// TIA Portal project "PLC_IHM" (V17)

(* hardware
DEVICE "HMI_1"  KTP400 Comfort
   slot 0: "HMI_1"  KTP400 Comfort  6AV2 124-2DC01-0AX0  16.0.0.0
   slot 1: "HMI_RT_1"  KTP400 Comfort  6AV2 124-2DC01-0AX0  16.0.0.0
   slot 5: "HMI_1.IE_CP_1"  PROFINET Interface  16.0.0.0
      slot 1: "PROFINET Interface_1"  PROFINET Interface
         slot 1: "Port_1"  Port
   slot 7: "HMI_1.MPI/DP_CP_1"  MPI/DP Interface  16.0.0.0
DEVICE "S7-1200 station_1"  S7-1200 Station
   slot 0: "Rack_0"  S7-1200 Rack  Rack  V1.0
   slot 1: "PLC_1"  CPU 1211C DC/DC/Rly  6ES7 211-1HE40-0XB0  V4.5
*)

// ===== PLC "PLC_1"  CPU 1211C DC/DC/Rly =====

VAR_GLOBAL   // PLC tag table "Default tag table"
   "Tag_1" AT %I0.0 : Bool;
   "Tag_3" AT %I0.1 : Bool;
   "Tag_5" AT %I0.2 : Bool;
   "Tag_8" AT %I0.3 : Bool;
   "Tag_9" AT %I0.4 : Bool;
   "CPLUS" AT %Q0.0 : Bool;
   "CMOINS" AT %Q0.1 : Bool;
   "MPLUS" AT %Q0.2 : Bool;
   "MMOINS" AT %Q0.3 : Bool;
   "IHM_TEST_Q0" AT %M0.0 : Bool;
   "IHM_TEST_Q1" AT %M0.1 : Bool;
   "IHM_TEST_Q2" AT %M0.2 : Bool;
   "IHM_TEST_Q3" AT %M0.3 : Bool;
   "X0" AT %M1.0 : Bool;
   "X2" AT %M1.1 : Bool;
   "X3" AT %M1.2 : Bool;
   "X4" AT %M1.3 : Bool;
   "X5" AT %M1.4 : Bool;
   "X6" AT %M1.5 : Bool;
   "X7" AT %M1.6 : Bool;
   "DCY" AT %M2.0 : Bool;
   "C1" AT %M2.1 : Bool;
   "C2" AT %M2.2 : Bool;
   "C3" AT %M2.3 : Bool;
   "DECHARGE" AT %M2.4 : Bool;
   "HAUT" AT %M2.5 : Bool;
   "BAS" AT %M2.6 : Bool;
   "X1" AT %M2.7 : Bool;
   "FIN_TEMPO" AT %M3.0 : Bool;
   "MOVE_X_PIECE" AT %MW20 : Int;
   "MOVE_Y_PIECE" AT %MW4 : Int;
   "SendInitParam" AT %M3.1 : Bool;
   "SendInitMemo" AT %M3.2 : Bool;
   "MOVE_X_CHARIOT" AT %MW6 : Int;
   "MOVE_Y_CHARIOT" AT %MW8 : Int;
   "MOVE_X_CORDON" AT %MW10 : Int;
   "MOVE_Y_CORDON" AT %MW12 : Int;
   "tempoTime" AT %MD30 : Time;
   "CompteurPiece" AT %MW24 : Int;
   "MemoI0" AT %M30.0 : Bool;
   "MemoI1" AT %M30.1 : Bool;
   "MemoI2" AT %M30.2 : Bool;
   "MemoI3" AT %M30.3 : Bool;
   "Tempo_Int_To_Time" AT %MD34 : Time;
   "Tempo_Int" AT %MW26 : Int;
   "Tempo_Time_To_Int" AT %MW28 : Int;
END_VAR

// folder: System blocks/Program resources

DATA_BLOCK "TEMPO"   // DB1
{ S7_Optimized_Access := 'TRUE' }
AUTHOR : Simatic
FAMILY : IEC
NAME : IEC_TMR
VERSION : 1.0
// stored: InstanceOfName IEC_TIMER
"IEC_TIMER"
BEGIN
END_DATA_BLOCK

// folder: (top level)

FUNCTION "TestInputOutput" : Void   // FC1, LAD
{ S7_Optimized_Access := 'TRUE' }
VERSION : 0.1
BEGIN

REGION Network 1: I0 alumme Q0
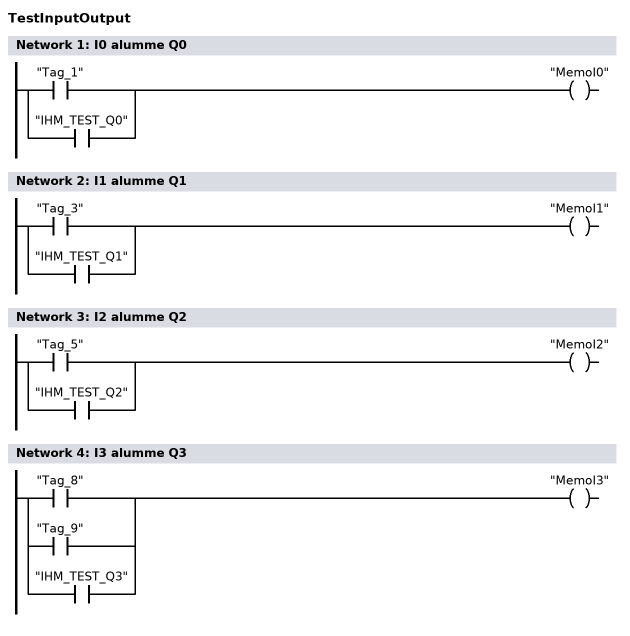
   RUNG wire#powerrail
      Contact( "Tag_1" )
      wire#w1
      Coil( "MemoI0" )
   END_RUNG
   RUNG wire#powerrail
      Contact( "IHM_TEST_Q0" )
   END_RUNG wire#w1
   // the same network as SCL:
   "MemoI0" := "Tag_1" OR "IHM_TEST_Q0";
END_REGION

REGION Network 2: I1 alumme Q1
   RUNG wire#powerrail
      Contact( "Tag_3" )
      wire#w1
      Coil( "MemoI1" )
   END_RUNG
   RUNG wire#powerrail
      Contact( "IHM_TEST_Q1" )
   END_RUNG wire#w1
   // the same network as SCL:
   "MemoI1" := "Tag_3" OR "IHM_TEST_Q1";
END_REGION

REGION Network 3: I2 alumme Q2
   RUNG wire#powerrail
      Contact( "Tag_5" )
      wire#w1
      Coil( "MemoI2" )
   END_RUNG
   RUNG wire#powerrail
      Contact( "IHM_TEST_Q2" )
   END_RUNG wire#w1
   // the same network as SCL:
   "MemoI2" := "Tag_5" OR "IHM_TEST_Q2";
END_REGION

REGION Network 4: I3 alumme Q3
   RUNG wire#powerrail
      Contact( "Tag_8" )
      wire#w1
      Coil( "MemoI3" )
   END_RUNG
   RUNG wire#powerrail
      Contact( "Tag_9" )
   END_RUNG wire#w1
   RUNG wire#powerrail
      Contact( "IHM_TEST_Q3" )
   END_RUNG wire#w1
   // the same network as SCL:
   "MemoI3" := "Tag_8" OR "Tag_9" OR "IHM_TEST_Q3";
END_REGION
END_FUNCTION

FUNCTION "BAIN_DEGRESSAGE" : Void   // FC2, LAD
{ S7_Optimized_Access := 'TRUE' }
VERSION : 0.1
BEGIN

REGION Network 1: X0
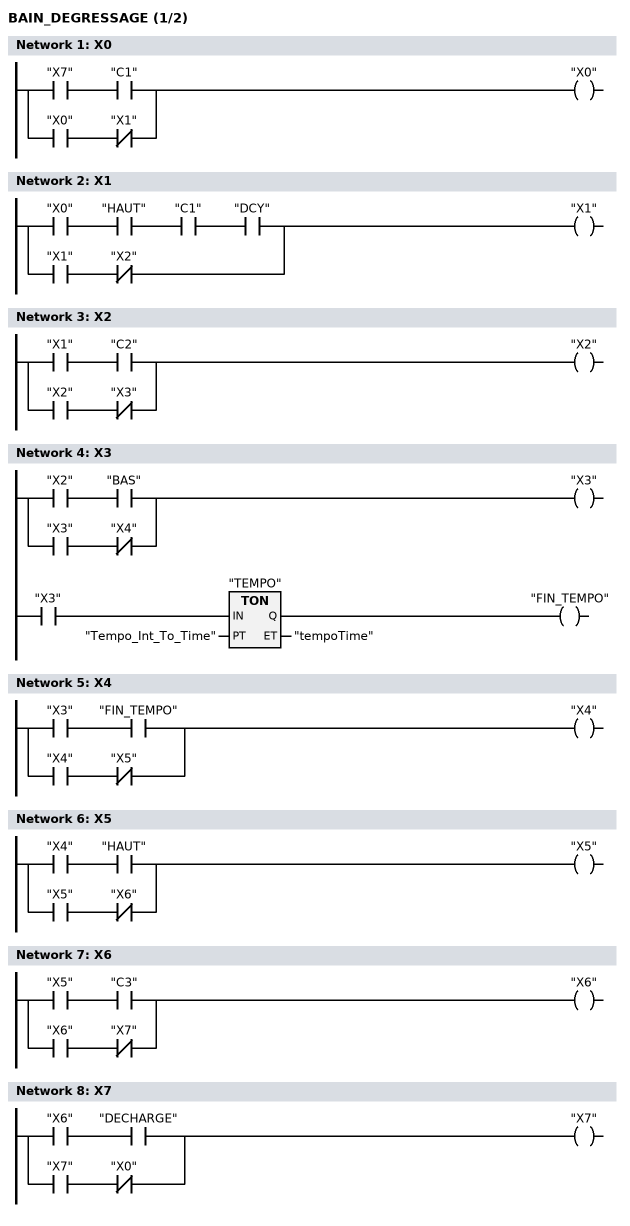
   RUNG wire#powerrail
      Contact( "X7" )
      Contact( "C1" )
      wire#w1
      Coil( "X0" )
   END_RUNG
   RUNG wire#powerrail
      Contact( "X0" )
      I_Contact( "X1" )
   END_RUNG wire#w1
   // the same network as SCL:
   "X0" := ("X7" AND "C1") OR ("X0" AND NOT "X1");
END_REGION

REGION Network 2: X1
   RUNG wire#powerrail
      Contact( "X0" )
      Contact( "HAUT" )
      Contact( "C1" )
      Contact( "DCY" )
      wire#w1
      Coil( "X1" )
   END_RUNG
   RUNG wire#powerrail
      Contact( "X1" )
      I_Contact( "X2" )
   END_RUNG wire#w1
   // the same network as SCL:
   "X1" := ("X0" AND "HAUT" AND "C1" AND "DCY") OR ("X1" AND NOT "X2");
END_REGION

REGION Network 3: X2
   RUNG wire#powerrail
      Contact( "X1" )
      Contact( "C2" )
      wire#w1
      Coil( "X2" )
   END_RUNG
   RUNG wire#powerrail
      Contact( "X2" )
      I_Contact( "X3" )
   END_RUNG wire#w1
   // the same network as SCL:
   "X2" := ("X1" AND "C2") OR ("X2" AND NOT "X3");
END_REGION

REGION Network 4: X3
   "X3" := ("X2" AND "BAS") OR ("X3" AND NOT "X4");
   "TEMPO".TON(IN := "X3", PT := "Tempo_Int_To_Time", ET => "tempoTime");
   "FIN_TEMPO" := "TEMPO".Q;
END_REGION

REGION Network 5: X4
   RUNG wire#powerrail
      Contact( "X3" )
      Contact( "FIN_TEMPO" )
      wire#w1
      Coil( "X4" )
   END_RUNG
   RUNG wire#powerrail
      Contact( "X4" )
      I_Contact( "X5" )
   END_RUNG wire#w1
   // the same network as SCL:
   "X4" := ("X3" AND "FIN_TEMPO") OR ("X4" AND NOT "X5");
END_REGION

REGION Network 6: X5
   RUNG wire#powerrail
      Contact( "X4" )
      Contact( "HAUT" )
      wire#w1
      Coil( "X5" )
   END_RUNG
   RUNG wire#powerrail
      Contact( "X5" )
      I_Contact( "X6" )
   END_RUNG wire#w1
   // the same network as SCL:
   "X5" := ("X4" AND "HAUT") OR ("X5" AND NOT "X6");
END_REGION

REGION Network 7: X6
   RUNG wire#powerrail
      Contact( "X5" )
      Contact( "C3" )
      wire#w1
      Coil( "X6" )
   END_RUNG
   RUNG wire#powerrail
      Contact( "X6" )
      I_Contact( "X7" )
   END_RUNG wire#w1
   // the same network as SCL:
   "X6" := ("X5" AND "C3") OR ("X6" AND NOT "X7");
END_REGION

REGION Network 8: X7
   RUNG wire#powerrail
      Contact( "X6" )
      Contact( "DECHARGE" )
      wire#w1
      Coil( "X7" )
   END_RUNG
   RUNG wire#powerrail
      Contact( "X7" )
      I_Contact( "X0" )
   END_RUNG wire#w1
   // the same network as SCL:
   "X7" := ("X6" AND "DECHARGE") OR ("X7" AND NOT "X0");
END_REGION

REGION Network 9: SORTIE CPLUS
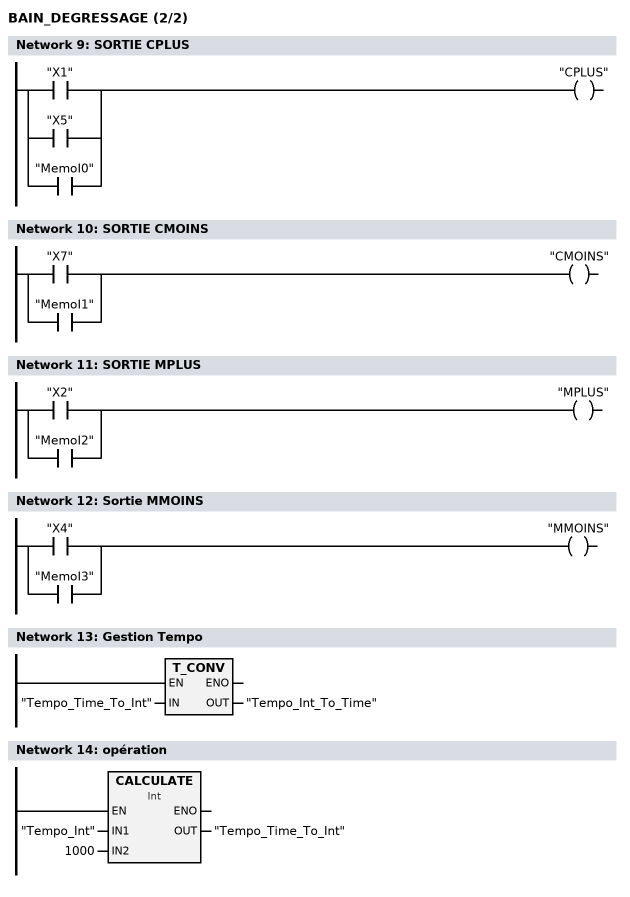
   RUNG wire#powerrail
      Contact( "X1" )
      wire#w1
      Coil( "CPLUS" )
   END_RUNG
   RUNG wire#powerrail
      Contact( "X5" )
   END_RUNG wire#w1
   RUNG wire#powerrail
      Contact( "MemoI0" )
   END_RUNG wire#w1
   // the same network as SCL:
   "CPLUS" := "X1" OR "X5" OR "MemoI0";
END_REGION

REGION Network 10: SORTIE CMOINS
   RUNG wire#powerrail
      Contact( "X7" )
      wire#w1
      Coil( "CMOINS" )
   END_RUNG
   RUNG wire#powerrail
      Contact( "MemoI1" )
   END_RUNG wire#w1
   // the same network as SCL:
   "CMOINS" := "X7" OR "MemoI1";
END_REGION

REGION Network 11: SORTIE MPLUS
   RUNG wire#powerrail
      Contact( "X2" )
      wire#w1
      Coil( "MPLUS" )
   END_RUNG
   RUNG wire#powerrail
      Contact( "MemoI2" )
   END_RUNG wire#w1
   // the same network as SCL:
   "MPLUS" := "X2" OR "MemoI2";
END_REGION

REGION Network 12: Sortie MMOINS
   RUNG wire#powerrail
      Contact( "X4" )
      wire#w1
      Coil( "MMOINS" )
   END_RUNG
   RUNG wire#powerrail
      Contact( "MemoI3" )
   END_RUNG wire#w1
   // the same network as SCL:
   "MMOINS" := "X4" OR "MemoI3";
END_REGION

REGION Network 13: Gestion Tempo
   "Tempo_Int_To_Time" := T_CONV(IN := "Tempo_Time_To_Int");
END_REGION

REGION Network 14: opération
   RUNG wire#powerrail
      { S7_Templates := "SrcType := Int"; S7_Expression := "IN1 * IN2" } Calculate(in1 := "Tempo_Int", in2 := 1000, out => "Tempo_Time_To_Int")
   END_RUNG
   // the same network as SCL:
   "Tempo_Time_To_Int" := "Tempo_Int" * 1000;
END_REGION
END_FUNCTION

FUNCTION "Maintenance" : Void   // FC3, LAD
{ S7_Optimized_Access := 'TRUE' }
VERSION : 0.1
BEGIN

REGION Network 1
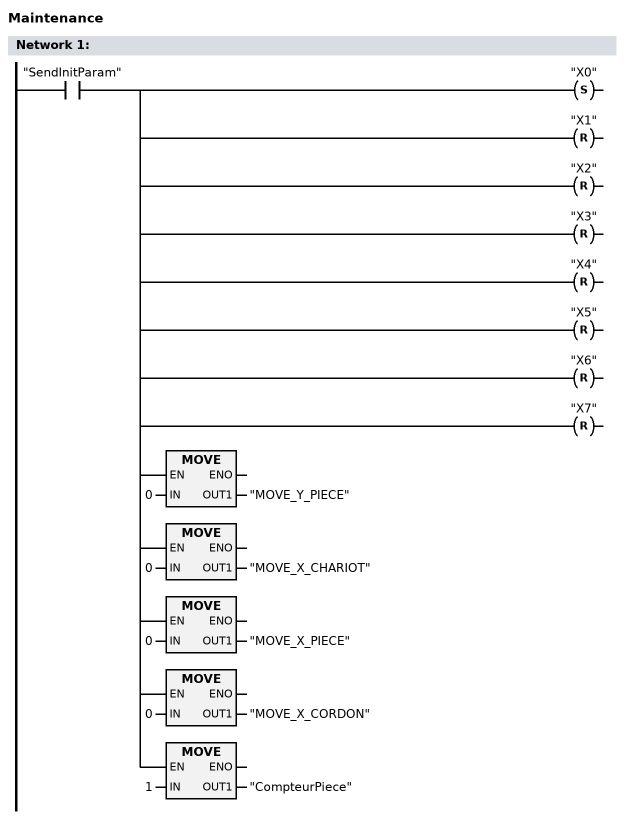
   RUNG wire#powerrail
      Contact( "SendInitParam" )
      wire#w1
      S_Coil( "X0" )
   END_RUNG
   RUNG wire#w1
      R_Coil( "X1" )
   END_RUNG
   RUNG wire#w1
      R_Coil( "X2" )
   END_RUNG
   RUNG wire#w1
      R_Coil( "X3" )
   END_RUNG
   RUNG wire#w1
      R_Coil( "X4" )
   END_RUNG
   RUNG wire#w1
      R_Coil( "X5" )
   END_RUNG
   RUNG wire#w1
      R_Coil( "X6" )
   END_RUNG
   RUNG wire#w1
      R_Coil( "X7" )
   END_RUNG
   RUNG wire#w1
      Move(in := 0, out1 => "MOVE_Y_PIECE")
   END_RUNG
   RUNG wire#w1
      Move(in := 0, out1 => "MOVE_X_CHARIOT")
   END_RUNG
   RUNG wire#w1
      Move(in := 0, out1 => "MOVE_X_PIECE")
   END_RUNG
   RUNG wire#w1
      Move(in := 0, out1 => "MOVE_X_CORDON")
   END_RUNG
   RUNG wire#w1
      Move(in := 1, out1 => "CompteurPiece")
   END_RUNG
   // the same network as SCL:
   IF "SendInitParam" THEN
       "X0" := TRUE;
       "X1" := FALSE;
       "X2" := FALSE;
       "X3" := FALSE;
       "X4" := FALSE;
       "X5" := FALSE;
       "X6" := FALSE;
       "X7" := FALSE;
       "MOVE_Y_PIECE" := 0;
       "MOVE_X_CHARIOT" := 0;
       "MOVE_X_PIECE" := 0;
       "MOVE_X_CORDON" := 0;
       "CompteurPiece" := 1;
   END_IF;
END_REGION
END_FUNCTION

ORGANIZATION_BLOCK "Main"   // OB1, LAD, ProgramCycle
TITLE = "Main Program Sweep (Cycle)"
{ S7_Optimized_Access := 'TRUE' }
VERSION : 0.1
   VAR_INPUT
      Initial_Call : Bool;   // Initial call of this OB
      Remanence : Bool;   // =True, if remanent data are available
   END_VAR
BEGIN

REGION Network 1: Test input output
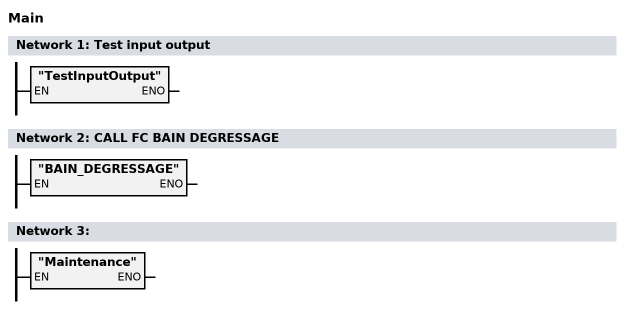
   RUNG wire#powerrail
      "TestInputOutput"()
   END_RUNG
   // the same network as SCL:
   "TestInputOutput"();
END_REGION

REGION Network 2: CALL FC BAIN DEGRESSAGE
   RUNG wire#powerrail
      "BAIN_DEGRESSAGE"()
   END_RUNG
   // the same network as SCL:
   "BAIN_DEGRESSAGE"();
END_REGION

REGION Network 3
   RUNG wire#powerrail
      "Maintenance"()
   END_RUNG
   // the same network as SCL:
   "Maintenance"();
END_REGION
END_ORGANIZATION_BLOCK

ORGANIZATION_BLOCK "Cyclic interrupt"   // OB30, LAD, CyclicInterrupt
{ S7_Optimized_Access := 'TRUE' }
VERSION : 0.1
   VAR_INPUT
      Initial_Call : Bool;   // Initial call of this OB
      Event_Count : Int;   // Events discarded
   END_VAR
   VAR_TEMP   // added for the SCL form of the ladder/FBD networks
      _w1 : Bool;
   END_VAR
BEGIN

REGION Network 1: X0 / X4
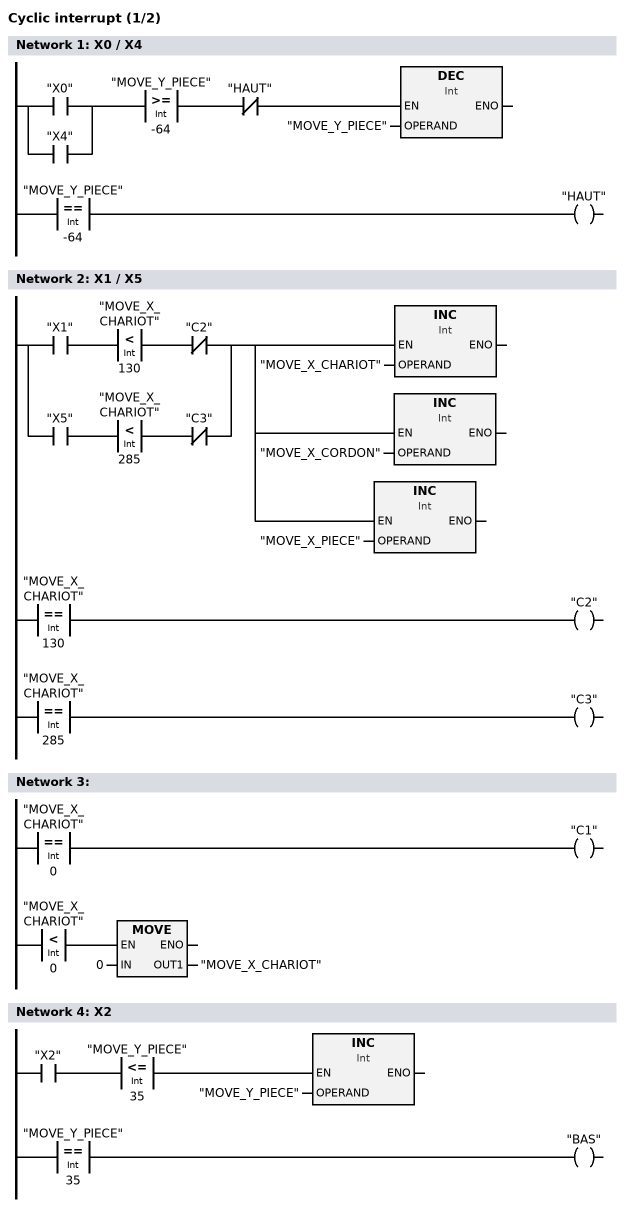
   RUNG wire#powerrail
      Contact( "X0" )
      wire#w1
      { S7_Templates := "SrcType := Int" } GE_Contact(in1 := "MOVE_Y_PIECE", in2 := -64)
      I_Contact( "HAUT" )
      { S7_Templates := "DestType := Int" } Dec( "MOVE_Y_PIECE" )
   END_RUNG
   RUNG wire#powerrail
      Contact( "X4" )
   END_RUNG wire#w1
   RUNG wire#powerrail
      { S7_Templates := "SrcType := Int" } EQ_Contact(in1 := "MOVE_Y_PIECE", in2 := -64)
      Coil( "HAUT" )
   END_RUNG
   // the same network as SCL:
   IF ("X0" OR "X4") AND ("MOVE_Y_PIECE" >= (-64)) AND NOT "HAUT" THEN
       "MOVE_Y_PIECE" := "MOVE_Y_PIECE" - 1;
   END_IF;
   "HAUT" := "MOVE_Y_PIECE" = (-64);
END_REGION

REGION Network 2: X1 / X5
   RUNG wire#powerrail
      Contact( "X1" )
      { S7_Templates := "SrcType := Int" } LT_Contact(in1 := "MOVE_X_CHARIOT", in2 := 130)
      I_Contact( "C2" )
      wire#w1
      { S7_Templates := "DestType := Int" } Inc( "MOVE_X_CHARIOT" )
   END_RUNG
   RUNG wire#powerrail
      Contact( "X5" )
      { S7_Templates := "SrcType := Int" } LT_Contact(in1 := "MOVE_X_CHARIOT", in2 := 285)
      I_Contact( "C3" )
   END_RUNG wire#w1
   RUNG wire#w1
      { S7_Templates := "DestType := Int" } Inc( "MOVE_X_CORDON" )
   END_RUNG
   RUNG wire#w1
      { S7_Templates := "DestType := Int" } Inc( "MOVE_X_PIECE" )
   END_RUNG
   RUNG wire#powerrail
      { S7_Templates := "SrcType := Int" } EQ_Contact(in1 := "MOVE_X_CHARIOT", in2 := 130)
      Coil( "C2" )
   END_RUNG
   RUNG wire#powerrail
      { S7_Templates := "SrcType := Int" } EQ_Contact(in1 := "MOVE_X_CHARIOT", in2 := 285)
      Coil( "C3" )
   END_RUNG
   // the same network as SCL:
   #_w1 := ("X1" AND ("MOVE_X_CHARIOT" < 130) AND NOT "C2") OR ("X5" AND ("MOVE_X_CHARIOT" < 285) AND NOT "C3");
   IF #_w1 THEN
       "MOVE_X_CHARIOT" := "MOVE_X_CHARIOT" + 1;
       "MOVE_X_CORDON" := "MOVE_X_CORDON" + 1;
       "MOVE_X_PIECE" := "MOVE_X_PIECE" + 1;
   END_IF;
   "C2" := "MOVE_X_CHARIOT" = 130;
   "C3" := "MOVE_X_CHARIOT" = 285;
END_REGION

REGION Network 3
   RUNG wire#powerrail
      { S7_Templates := "SrcType := Int" } EQ_Contact(in1 := "MOVE_X_CHARIOT", in2 := 0)
      Coil( "C1" )
   END_RUNG
   RUNG wire#powerrail
      { S7_Templates := "SrcType := Int" } LT_Contact(in1 := "MOVE_X_CHARIOT", in2 := 0)
      Move(in := 0, out1 => "MOVE_X_CHARIOT")
   END_RUNG
   // the same network as SCL:
   "C1" := "MOVE_X_CHARIOT" = 0;
   IF "MOVE_X_CHARIOT" < 0 THEN "MOVE_X_CHARIOT" := 0; END_IF;
END_REGION

REGION Network 4: X2
   RUNG wire#powerrail
      Contact( "X2" )
      { S7_Templates := "SrcType := Int" } LE_Contact(in1 := "MOVE_Y_PIECE", in2 := 35)
      { S7_Templates := "DestType := Int" } Inc( "MOVE_Y_PIECE" )
   END_RUNG
   RUNG wire#powerrail
      { S7_Templates := "SrcType := Int" } EQ_Contact(in1 := "MOVE_Y_PIECE", in2 := 35)
      Coil( "BAS" )
   END_RUNG
   // the same network as SCL:
   IF "X2" AND ("MOVE_Y_PIECE" <= 35) THEN "MOVE_Y_PIECE" := "MOVE_Y_PIECE" + 1; END_IF;
   "BAS" := "MOVE_Y_PIECE" = 35;
END_REGION

REGION Network 5: X7
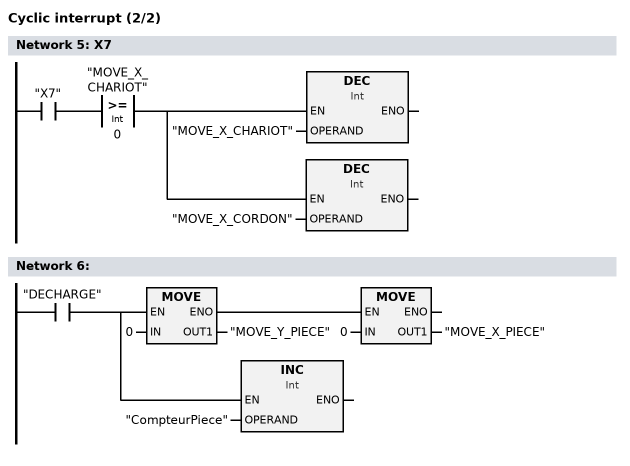
   RUNG wire#powerrail
      Contact( "X7" )
      { S7_Templates := "SrcType := Int" } GE_Contact(in1 := "MOVE_X_CHARIOT", in2 := 0)
      wire#w1
      { S7_Templates := "DestType := Int" } Dec( "MOVE_X_CHARIOT" )
   END_RUNG
   RUNG wire#w1
      { S7_Templates := "DestType := Int" } Dec( "MOVE_X_CORDON" )
   END_RUNG
   // the same network as SCL:
   #_w1 := "X7" AND ("MOVE_X_CHARIOT" >= 0);
   IF #_w1 THEN
       "MOVE_X_CHARIOT" := "MOVE_X_CHARIOT" - 1;
       "MOVE_X_CORDON" := "MOVE_X_CORDON" - 1;
   END_IF;
END_REGION

REGION Network 6
   RUNG wire#powerrail
      Contact( "DECHARGE" )
      wire#w1
      Move(in := 0, out1 => "MOVE_Y_PIECE")
      Move(in := 0, out1 => "MOVE_X_PIECE")
   END_RUNG
   RUNG wire#w1
      { S7_Templates := "DestType := Int" } Inc( "CompteurPiece" )
   END_RUNG
   // the same network as SCL:
   IF "DECHARGE" THEN
       "MOVE_Y_PIECE" := 0;
       "MOVE_X_PIECE" := 0;
       "CompteurPiece" := "CompteurPiece" + 1;
   END_IF;
END_REGION
END_ORGANIZATION_BLOCK

(* ===== HMI "HMI_RT_1" =====
system functions are stored by id; their names below are inferred from use
connection "HMI_Connection_1": ETHERNET, S7_1200_OMS

HMI tags "Default tag table"
   "Tag_ScreenNumber" : UInt, internal
   "IHM_TEST_Q0" : Bool, internal
   "IHM_TEST_Q1" : Bool, internal
   "IHM_TEST_Q2" : Bool, internal
   "IHM_TEST_Q3" : Bool, internal
   "IHM_TEST_Q0(1)" : Bool = PLC IHM_TEST_Q0 AT %M0.0, 1 s
   "IHM_TEST_Q1(1)" : Bool = PLC IHM_TEST_Q1 AT %M0.1, 1 s
   "IHM_TEST_Q2(1)" : Bool = PLC IHM_TEST_Q2 AT %M0.2, 1 s
   "IHM_TEST_Q3(1)" : Bool = PLC IHM_TEST_Q3 AT %M0.3, 1 s
   "X0" : Bool = PLC X0 AT %M1.0, 1 s
   "X1" : Bool = PLC X1 AT %M2.7, 1 s
   "X2" : Bool = PLC X2 AT %M1.1, 1 s
   "X3" : Bool = PLC X3 AT %M1.2, 1 s
   "X4" : Bool = PLC X4 AT %M1.3, 1 s
   "X5" : Bool = PLC X5 AT %M1.4, 1 s
   "X6" : Bool = PLC X6 AT %M1.5, 1 s
   "X7" : Bool = PLC X7 AT %M1.6, 1 s
   "HAUT" : Bool = PLC HAUT AT %M2.5, 1 s
   "BAS" : Bool = PLC BAS AT %M2.6, 1 s
   "C1" : Bool = PLC C1 AT %M2.1, 1 s
   "C2" : Bool = PLC C2 AT %M2.2, 1 s
   "C3" : Bool = PLC C3 AT %M2.3, 1 s
   "DCY" : Bool = PLC DCY AT %M2.0, 1 s
   "DECHARGE" : Bool = PLC DECHARGE AT %M2.4, 1 s
   "MOVE_Y_PIECE" : Int = PLC MOVE_Y_PIECE AT %MW4, 1 s
   "MOVE_X_PIECE" : Int = PLC MOVE_X_PIECE AT %MW20, 1 s
   "MOVE_Y_CHARIOT" : Int = PLC MOVE_Y_CHARIOT AT %MW8, 1 s
   "MOVE_X_CHARIOT(1)" : Int = PLC MOVE_X_CHARIOT AT %MW6, 1 s
   "SendInitParam" : Bool = PLC SendInitParam AT %M3.1, 1 s
   "MOVE_X_CORDON" : Int = PLC MOVE_X_CORDON AT %MW10, 1 s
   "MOVE_Y_CORDON" : Int = PLC MOVE_Y_CORDON AT %MW12, 1 s
   "tempoTime" : Time = PLC tempoTime AT %MD30, 1 s
   "CompteurPiece" : Int = PLC CompteurPiece AT %MW24, 1 s
   "Tempo_Int" : Int = PLC Tempo_Int AT %MW26, 1 s

screen "Root screen" 480x272, template "Template_1"
   on GenerateScreen: SetTag("Tag_ScreenNumber", 1)
   Button "Button_1" at 11,13 size 139x32; TextOff 'VUE TEST OUTPUT'
      on Click: ActivateScreen("TEST_OUTPUT", 0)
   Button "Button_2" at 165,13 size 139x32; TextOff 'VUE GRAFCET'
      on Click: ActivateScreen("GRAFCET", 0)
   Button "Button_3" at 326,13 size 139x32; TextOff 'VUE SYSTEME'
      on Click: ActivateScreen("SYTEME DEGRESSAGE", 0)
   Button "Button_4" at 11,74 size 139x32; TextOff 'VUE MAINTENANCE'
      on Click: ActivateScreen("Maintenance", 0)
   Softkey "Softkey_F4" at 0,0 size 0x0
      on KeyDown: ActivateScreen("Maintenance", 0)
   Softkey "Softkey_F3" at 0,0 size 0x0
      on KeyDown: ActivateScreen("TEST_OUTPUT", 0)
   Softkey "Softkey_F1" at 0,0 size 0x0
      on KeyDown: ActivateScreen("GRAFCET", 0)
   Softkey "Softkey_F2" at 0,0 size 0x0
      on KeyDown: ActivateScreen("SYTEME DEGRESSAGE", 0)

Template "Template_1" 480x272
   Button "Exit" at 379,148 size 63x63; TextOff 'Exit'; PictureOff "ExitRuntime_KTP400_Comfort_TR"; PictureOn "ExitRuntime_KTP400_Comfort_TR"
      on Release: StopRuntime(0)
   Button "Template_Button" at 265,148 size 63x63; TextOff 'Text'
   Button "Alarms" at 151,148 size 63x63; TextOff 'Alarms'; PictureOff "AlarmDisplay_KTP400_Comfort_TR"; PictureOn "AlarmDisplay_KTP400_Comfort_TR"
      on Release: function_ef3f5d25("Alarm window_Unacknowledged", -1)
   Button "Start screen" at 37,148 size 63x63; TextOff 'Start screen'; PictureOff "NavigateHome_KTP400_Comfort_TR"; PictureOn "NavigateHome_KTP400_Comfort_TR"
      on Release: ActivateScreen("Root screen", 0)

screen "TEST_OUTPUT" 480x272
   Button "Button_1" at 26,19 size 96x32; TextOff '%Q0.0'
      on Click: InvertBit("IHM_TEST_Q0(1)")
   Button "Button_2" at 134,19 size 96x32; TextOff '%Q0.1'
      on Click: InvertBit("IHM_TEST_Q1(1)")
   Button "Button_3" at 242,19 size 96x32; TextOff '%Q0.2'
      on Click: InvertBit("IHM_TEST_Q2(1)")
   Button "Button_4" at 350,19 size 96x32; TextOff '%Q0.3'
      on Click: InvertBit("IHM_TEST_Q3(1)")
   Button "Button_5" at 173,173 size 96x32; TextOff 'Back Home'
      on Click: ActivateScreen("Root screen", 0)
   Circle "Circle_1" at 51,61 size 48x48
      Appearance <- "IHM_TEST_Q0(1)"
   Circle "Circle_2" at 154,60 size 48x48
      Appearance <- "IHM_TEST_Q1(1)"
   Circle "Circle_3" at 257,59 size 48x48
      Appearance <- "IHM_TEST_Q2(1)"
   Circle "Circle_4" at 360,58 size 48x48
      Appearance <- "IHM_TEST_Q3(1)"

screen "GRAFCET" 480x272
   Rectangle "Rectangle_2" at 57,161 size 50x50
      Appearance <- "X1"
   Rectangle "Rectangle_3" at 155,60 size 50x50
      Appearance <- "X2"
   Rectangle "Rectangle_4" at 155,160 size 50x50
      Appearance <- "X3"
   Rectangle "Rectangle_5" at 255,60 size 50x50
      Appearance <- "X4"
   Rectangle "Rectangle_6" at 255,160 size 50x50
      Appearance <- "X5"
   Rectangle "Rectangle_7" at 357,60 size 50x50
      Appearance <- "X6"
   Rectangle "Rectangle_8" at 357,160 size 50x50
      Appearance <- "X7"
   Button "Button_1" at 376,8 size 96x32; TextOff 'VUE HOME'
      on Click: ActivateScreen("Root screen", 0)
   TextField "Text field_2" at 64,176 size 24x20; Text 'X1'
   TextField "Text field_3" at 167,75 size 24x20; Text 'X2'
   TextField "Text field_4" at 165,179 size 24x20; Text 'X3'
   TextField "Text field_5" at 266,75 size 24x20; Text 'X4'
   TextField "Text field_6" at 269,175 size 24x20; Text 'X5'
   TextField "Text field_7" at 373,73 size 24x20; Text 'X6'
   TextField "Text field_8" at 372,176 size 24x20; Text 'X7'
   Button "Button_2" at 306,122 size 40x30; TextOff 'H'
      on Press: SetBit("HAUT")
      on Release: ResetBit("HAUT")
   Button "Button_3" at 2,14 size 34x29; TextOff 'DCY'
      on Press: SetBit("DCY")
      on Release: ResetBit("DCY")
   Button "Button_4" at 106,223 size 40x30; TextOff 'C2'
      on Press: SetBit("C2")
      on Release: ResetBit("C2")
   Button "Button_5" at 205,120 size 40x30; TextOff 'B'
      on Press: SetBit("BAS")
      on Release: ResetBit("BAS")
   Button "Button_6" at 206,222 size 40x30; TextOff 'T'
   Button "Button_7" at 105,122 size 40x30; TextOff 'H'
      on Press: SetBit("HAUT")
      on Release: ResetBit("HAUT")
   Button "Button_8" at 306,222 size 40x30; TextOff 'C3'
      on Press: SetBit("C3")
      on Release: ResetBit("C3")
   Button "Button_9" at 406,120 size 40x30; TextOff 'D'
      on Release: ResetBit("DECHARGE")
      on Press: SetBit("DECHARGE")
   Rectangle "Rectangle_1" at 54,60 size 50x50
      Appearance <- "X0"
   Button "Button_10" at 25,121 size 40x30; TextOff 'C1'
      on Press: SetBit("C1")
      on Release: ResetBit("C1")
   TextField "Text field_9" at 66,77 size 24x20; Text 'X0'
   Button "Button_11" at 405,223 size 40x30; TextOff 'C1'
      on Release: ResetBit("C1")
      on Press: SetBit("C1")
   Softkey "Softkey_F1" at 0,0 size 0x0
      on KeyDown: ActivateScreen("SYTEME DEGRESSAGE", 0)

screen "SYTEME DEGRESSAGE" 480x272
   Button "Button_1" at 383,253 size 96x19; TextOff 'VUE HOME'
      on Click: ActivateScreen("Root screen", 0)
   Group "Group_1" at 82,18 size 38x33
   Group "Group_2" at 234,18 size 38x33
   Group "Group_3" at 386,18 size 38x33
   Button "Button_2" at 0,119 size 42x26; TextOff 'DCY'
      on Press: SetBit("DCY")
      on Release: ResetBit("DCY")
   Button "Button_3" at 438,112 size 42x26; TextOff 'DCH'
      on Press: SetBit("DECHARGE")
      on Release: ResetBit("DECHARGE")
   Line "Line_52" at 106,69 size 1x88
      DirectMovement <- "MOVE_X_CORDON"
      DirectMovement <- "MOVE_Y_CORDON"
   TextField "Text field_1" at 87,15 size 23x20; Text 'C1'
   TextField "Text field_2" at 238,16 size 23x20; Text 'C2'
   TextField "Text field_3" at 389,16 size 23x20; Text 'C3'
   Circle "Circle_6" at 229,244 size 14x14
      Appearance <- "BAS"
   Group "Group_5" at 50,47 size 126x52
      DirectMovement <- "MOVE_Y_CHARIOT"
      DirectMovement <- "MOVE_X_CHARIOT(1)"
   Button "Button_4" at 0,240 size 124x32; TextOff 'Send init Param'
      on Release: ResetBit("SendInitParam")
      on Press: SetBit("SendInitParam")
   IOField "I/O field_1" at 376,217 size 85x32; FormatPattern 999999
      ProcessValue <- "tempoTime"
   Group "Group_6" at 77,158 size 58x51
   IOField "Champ d'E/S_1" at 376,151 size 96x32; FormatPattern 99999
      ProcessValue <- "Tempo_Int"
   Circle "Circle_1" at 106,37 size 14x14
      Appearance <- "C1"
   Group "Group" at 50,47 size 126x38
   Circle "Circle_7" at 127,90 size 9x9
      Appearance <- "HAUT"
   Rectangle "Rectangle_9" at 77,158 size 58x51
      DirectMovement <- "MOVE_X_PIECE"
      DirectMovement <- "MOVE_Y_PIECE"
   IOField "I/O field_2" at 93,166 size 28x31; FormatPattern 99
      ProcessValue <- "CompteurPiece"
      DirectMovement <- "MOVE_X_PIECE"
      DirectMovement <- "MOVE_Y_PIECE"
   Circle "Circle_2" at 258,37 size 14x14
      Appearance <- "C2"
   Circle "Circle_3" at 410,37 size 14x14
      Appearance <- "C3"
   Group "Group_4" at 50,47 size 126x52
   Softkey "Softkey_F1" at 0,0 size 0x0
      on KeyDown: ActivateScreen("GRAFCET", 0)

screen "Maintenance" 480x272
   Button "Button_1" at 382,238 size 96x32; TextOff 'vue home'
      on Click: ActivateScreen("Root screen", 0)
   Button "Button_2" at 10,8 size 124x32; TextOff 'Send init Param'
      on Press: SetBit("SendInitParam")
      on Release: ResetBit("SendInitParam")
*)